# EPICS StreamDevice protocol: apps/keithleyApp/Db/keithley2001.proto
OutTerminator = LF;
InTerminator = LF;
ExtraInput = Ignore;

# units = milliseconds
WriteTimeout = 500;
ReadTimeout = 5000;
ReplyTimeout = 5000;

cmd       { out "\$1"; }

putInt    { out "\$1 %d"; @init { wait 100; out "\$1?"; in "%d"; } }
putFloat  { out "\$1 %f"; @init { wait 100; out "\$1?"; in "%f"; } }
putString { out "\$1 %s"; @init { wait 100; out "\$1?"; in "%s"; } }

getInt    { out "\$1?"; in "%d"; }
getFloat  { out "\$1?"; in "%f"; }
getString { out "\$1?"; in "%#s"; }
pressKey  { out ":SYST:KEY \$1"; }

getData {
    separator = ",";
    out ":TRAC:DATA?";
    in "%E";
#    @mismatch { in "%*s"; }
}

trigger2 {
    # enter key:
    out ":SYST:KEY 18";
    # trigger key:
    out ":SYST:KEY 30";
}

reset {
    out "*RST";
    wait 100;
    out ":SYST:PRES";
    wait 100;
    out ":STAT:PRES";
    wait 100;
    out ":ABOR";
    wait 100;
    out "*CLS";
    wait 100;
    out "*WAI";
    wait 100;
}
